{attribute 'linkalways'} 
{attribute 'no_explicit_call' := 'This FB is a CLASS and must be accessed using methods or properties'}
{attribute 'enable_dynamic_creation'}
FUNCTION_BLOCK PUBLIC DefaultMotionBuilder IMPLEMENTS MotionBuilder
VAR
	parameters : BuilderParameters;
	move_builder : DefaultMoveBuilder(parent_builder := THIS^, parameters := parameters);
	move_velocity_builder : DefaultMoveVelocityBuilder(parent_builder := THIS^, parameters := parameters);
	move_absolute_builder : DefaultMoveAbsoluteBuilder(parent_builder := THIS^, parameters := parameters);
	move_relative_builder : DefaultMoveRelativeBuilder(parent_builder := THIS^, parameters := parameters);
	gear_in_builder : DefaultGearInBuilder(parent_builder := THIS^, parameters := parameters);
END_VAR

METHOD PUBLIC Acceleration : MoveBuilder
VAR_INPUT
	value : LREAL;
END_VAR
parameters.acceleration := value;
Acceleration := move_builder;
END_METHOD

METHOD PUBLIC BufferMode : MoveBuilder
VAR_INPUT
	mode : MotionBufferMode;
END_VAR
parameters.buffer_mode := mode;
BufferMode := move_builder;
END_METHOD

METHOD PUBLIC BuildGearOutCommand : AsyncCommand
VAR_INPUT
	axis : REFERENCE TO Mc2Axis;
END_VAR
VAR
	command_ptr : POINTER TO GearOutCommand;
	command : AsyncCommand;
END_VAR
command_ptr := __NEW(GearOutCommand(
	axis := axis
));
BuildGearOutCommand := command_ptr^;
END_METHOD

METHOD PUBLIC BuildHaltCommand : MotionCommand
VAR_INPUT
	axis : REFERENCE TO Mc2Axis;
END_VAR
VAR
	command_ptr : POINTER TO HaltCommand;
	command : MotionCommand;
END_VAR
command_ptr := __NEW(HaltCommand(
	axis := axis,
	deceleration := parameters.deceleration,
	jerk := parameters.jerk,
	buffer_mode := parameters.buffer_mode
));
BuildHaltCommand := command_ptr^;
END_METHOD

METHOD PUBLIC BuildStopCommand : MotionCommand
VAR_INPUT
	axis : REFERENCE TO Mc2Axis;
END_VAR
VAR
	command_ptr : POINTER TO StopCommand;
	command : MotionCommand;
END_VAR
command_ptr := __NEW(StopCommand(
	axis := axis,
	deceleration := parameters.deceleration,
	jerk := parameters.jerk
));
BuildStopCommand := command_ptr^;
END_METHOD

METHOD PUBLIC Deceleration : MotionBuilder
VAR_INPUT
	value : LREAL;
END_VAR
parameters.deceleration := value;
Deceleration := THIS^;
END_METHOD

METHOD PUBLIC Distance : MoveRelativeBuilder
VAR_INPUT
	value : LREAL;
END_VAR
parameters.distance := value;
Distance := move_relative_builder;
END_METHOD

METHOD PUBLIC Jerk : MotionBuilder
VAR_INPUT
	value : LREAL;
END_VAR
parameters.jerk := value;
Jerk := THIS^;
END_METHOD

METHOD PUBLIC Position : MoveAbsoluteBuilder
VAR_INPUT
	value : LREAL;
END_VAR
parameters.position := value;
Position := move_absolute_builder;
END_METHOD

METHOD PUBLIC RatioDenominator : GearInBuilder
VAR_INPUT
	value : UINT;
END_VAR
parameters.ratio_denominator := value;
RatioDenominator := gear_in_builder;
END_METHOD

METHOD PUBLIC RatioNumerator : GearInBuilder
VAR_INPUT
	value : LREAL;
END_VAR
parameters.ratio_numerator := value;
RatioNumerator := gear_in_builder;
END_METHOD

METHOD PUBLIC Reset : MotionBuilder
parameters.acceleration := 0;
parameters.deceleration := 0;
parameters.jerk := 0;
parameters.buffer_mode := MotionBufferMode.Aborting;
Reset := THIS^;
END_METHOD

METHOD PUBLIC Velocity : MoveVelocityBuilder
VAR_INPUT
	value : LREAL;
END_VAR
parameters.velocity := value;
Velocity := move_velocity_builder;
END_METHOD

END_FUNCTION_BLOCK

(* stored: Version 1.1.0.1
   POU DefaultMotionBuilder: Id {a2edf869-84c6-0db6-0085-e9eeeeb63c74}, SpecialFunc None
   Folder Builders: Id {71879d48-47e6-0cab-387a-5d67b61154a0}
   Folder Property Setters: Id {ad35ec2c-16b4-0b94-3cac-7af0eeffa3a2}
   Method Acceleration: Id {e3e77b4e-beaf-08fb-2cc2-0b24bea83d64}
   Method BufferMode: Id {06ea8e4a-9a6b-04d6-268a-1a80b8fb3ff5}
   Method BuildGearOutCommand: Id {26b3a5cc-7687-4035-8ab6-99494cf1263a}
   Method BuildHaltCommand: Id {7b53665c-7b19-43e0-b1df-ec08ab259a79}
   Method BuildStopCommand: Id {7e9a74f9-4d3a-430e-a63e-10bb94b62f70}
   Method Deceleration: Id {a0d39c27-e434-07f5-15fa-bdfcb8b9862f}
   Method Distance: Id {a4c80f52-31d0-0c12-1ba3-af4dbc20b8b1}
   Method Jerk: Id {dd5b428f-4ff4-025d-0b10-09c472252f90}
   Method Position: Id {fe2fd08e-0eb0-0a47-0285-dd28cacda8d3}
   Method RatioDenominator: Id {71d0dac4-7e25-4e26-b773-671a618249c6}
   Method RatioNumerator: Id {59819601-f71a-4ef4-afd6-a659e26838c4}
   Method Reset: Id {22b5d9a1-b16c-02f7-3dfe-7e6088649161}
   Method Velocity: Id {3548811d-ee50-01f2-3562-7d2324338261} *)
